(* Logix 5000 project; controller Generic 1768-L43 rev 15.6; software revision 15.01; part 3 of 10 *)
(* tags used below, declared in another part *)
   EL_CTRL_5 : UDT_AxisHistory_CTRL;
   EL_CTRL_6 : UDT_AxisHistory_CTRL;
   EventLog_N5 : UDT_AxisHistory_DLM[51];
   EventLog_N6 : UDT_AxisHistory_DLM[51];
   LogLength : DINT;
   Motion_Group : ALIAS FOR MotionGroup;
   Servo_Axis_Node_5 : ALIAS FOR AXIS_Servo_Generic;
   Servo_Axis_Node_6 : ALIAS FOR AXIS_Servo_Generic;
(* AXIS_EventLog, continued *)

ROUTINE R05_EventLog_Node5   (* ladder *)
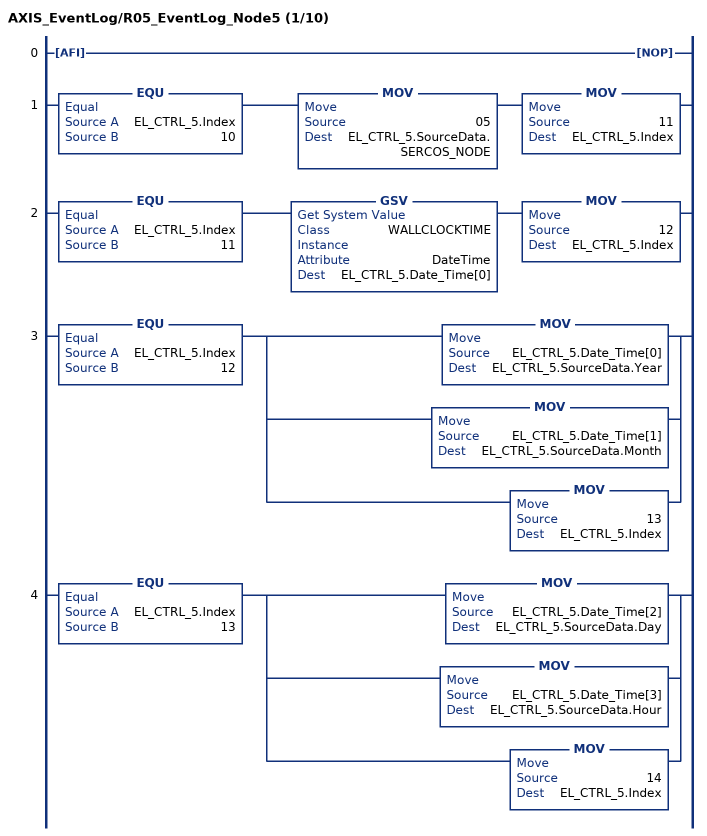
   0: AFI()NOP();
   1: EQU(EL_CTRL_5.Index,10)MOV(05,EL_CTRL_5.SourceData.SERCOS_NODE)MOV(11,EL_CTRL_5.Index);
   2: EQU(EL_CTRL_5.Index,11)GSV(WALLCLOCKTIME,,DateTime,EL_CTRL_5.Date_Time[0])MOV(12,EL_CTRL_5.Index);
   3: EQU(EL_CTRL_5.Index,12)[MOV(EL_CTRL_5.Date_Time[0],EL_CTRL_5.SourceData.Year) ,MOV(EL_CTRL_5.Date_Time[1],EL_CTRL_5.SourceData.Month) ,MOV(13,EL_CTRL_5.Index) ];
   4: EQU(EL_CTRL_5.Index,13)[MOV(EL_CTRL_5.Date_Time[2],EL_CTRL_5.SourceData.Day) ,MOV(EL_CTRL_5.Date_Time[3],EL_CTRL_5.SourceData.Hour) ,MOV(14,EL_CTRL_5.Index) ];
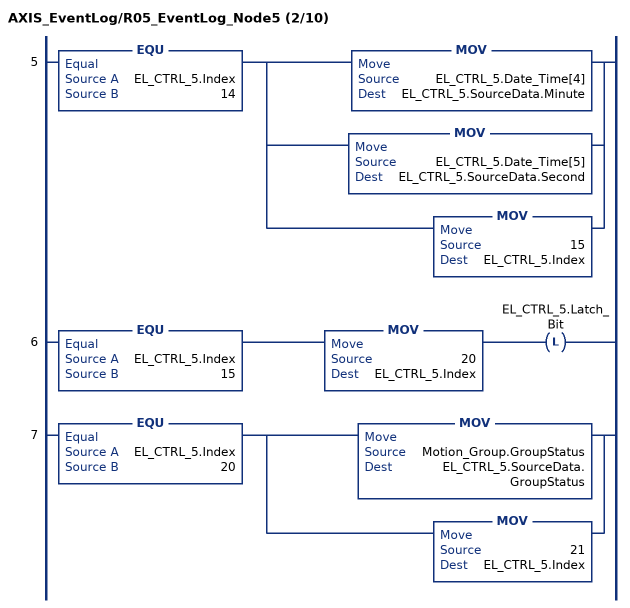
   5: EQU(EL_CTRL_5.Index,14)[MOV(EL_CTRL_5.Date_Time[4],EL_CTRL_5.SourceData.Minute) ,MOV(EL_CTRL_5.Date_Time[5],EL_CTRL_5.SourceData.Second) ,MOV(15,EL_CTRL_5.Index) ];
   6: EQU(EL_CTRL_5.Index,15)MOV(20,EL_CTRL_5.Index)OTL(EL_CTRL_5.Latch_Bit);
   7: EQU(EL_CTRL_5.Index,20)[MOV(Motion_Group.GroupStatus,EL_CTRL_5.SourceData.GroupStatus) ,MOV(21,EL_CTRL_5.Index) ];
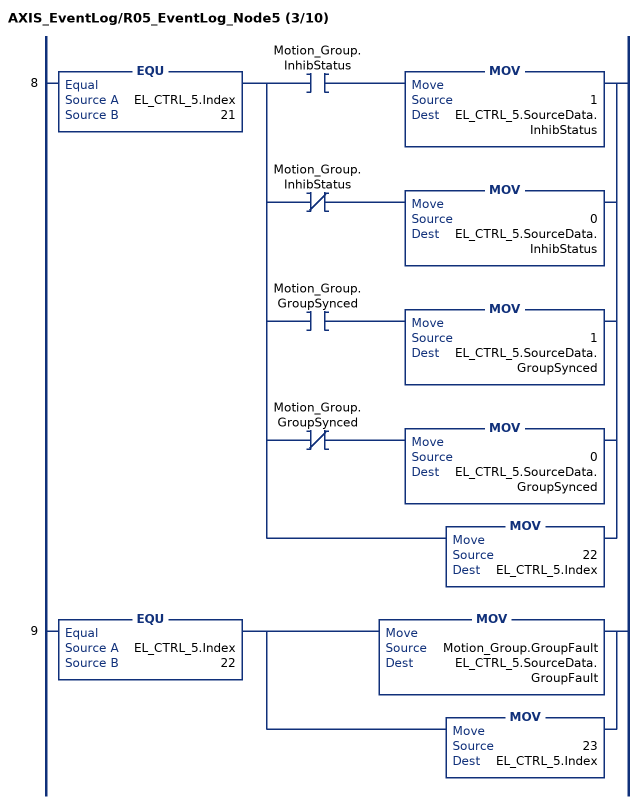
   8: EQU(EL_CTRL_5.Index,21)[XIC(Motion_Group.InhibStatus) MOV(1,EL_CTRL_5.SourceData.InhibStatus) ,XIO(Motion_Group.InhibStatus) MOV(0,EL_CTRL_5.SourceData.InhibStatus) ,XIC(Motion_Group.GroupSynced) MOV(1,EL_CTRL_5.SourceData.GroupSynced) ,XIO(Motion_Group.GroupSynced) MOV(0,EL_CTRL_5.SourceData.GroupSynced) ,MOV(22,EL_CTRL_5.Index) ];
   9: EQU(EL_CTRL_5.Index,22)[MOV(Motion_Group.GroupFault,EL_CTRL_5.SourceData.GroupFault) ,MOV(23,EL_CTRL_5.Index) ];
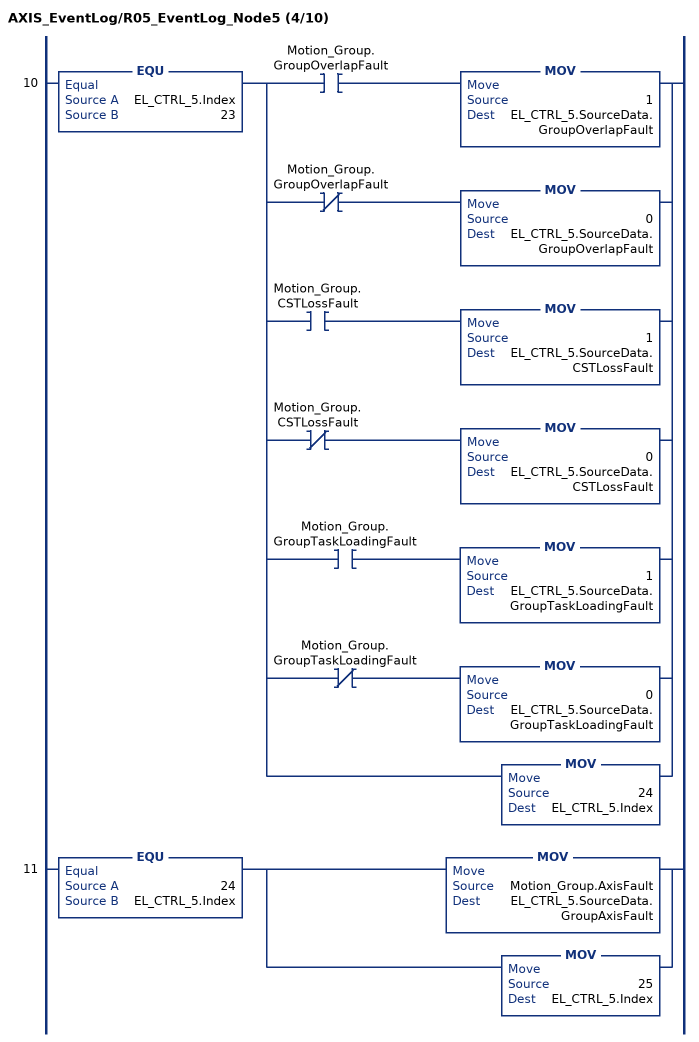
   10: EQU(EL_CTRL_5.Index,23)[XIC(Motion_Group.GroupOverlapFault) MOV(1,EL_CTRL_5.SourceData.GroupOverlapFault) ,XIO(Motion_Group.GroupOverlapFault) MOV(0,EL_CTRL_5.SourceData.GroupOverlapFault) ,XIC(Motion_Group.CSTLossFault) MOV(1,EL_CTRL_5.SourceData.CSTLossFault) ,XIO(Motion_Group.CSTLossFault) MOV(0,EL_CTRL_5.SourceData.CSTLossFault) ,XIC(Motion_Group.GroupTaskLoadingFault) MOV(1,EL_CTRL_5.SourceData.GroupTaskLoadingFault) ,XIO(Motion_Group.GroupTaskLoadingFault) MOV(0,EL_CTRL_5.SourceData.GroupTaskLoadingFault) ,MOV(24,EL_CTRL_5.Index) ];
   11: EQU(24,EL_CTRL_5.Index)[MOV(Motion_Group.AxisFault,EL_CTRL_5.SourceData.GroupAxisFault) ,MOV(25,EL_CTRL_5.Index) ];
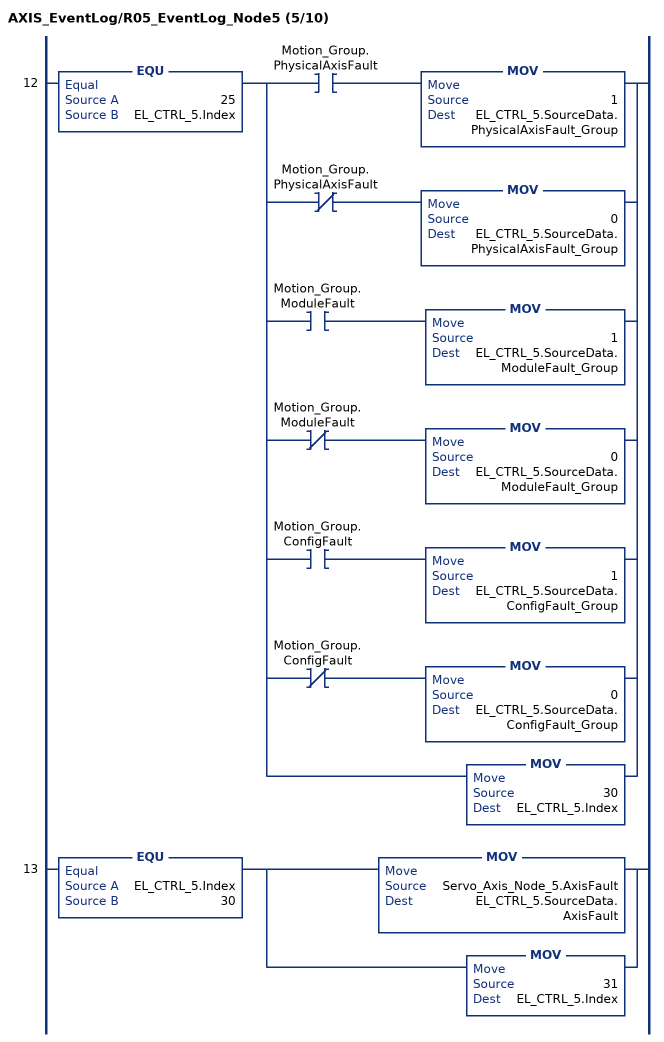
   12: EQU(25,EL_CTRL_5.Index)[XIC(Motion_Group.PhysicalAxisFault) MOV(1,EL_CTRL_5.SourceData.PhysicalAxisFault_Group) ,XIO(Motion_Group.PhysicalAxisFault) MOV(0,EL_CTRL_5.SourceData.PhysicalAxisFault_Group) ,XIC(Motion_Group.ModuleFault) MOV(1,EL_CTRL_5.SourceData.ModuleFault_Group) ,XIO(Motion_Group.ModuleFault) MOV(0,EL_CTRL_5.SourceData.ModuleFault_Group) ,XIC(Motion_Group.ConfigFault) MOV(1,EL_CTRL_5.SourceData.ConfigFault_Group) ,XIO(Motion_Group.ConfigFault) MOV(0,EL_CTRL_5.SourceData.ConfigFault_Group) ,MOV(30,EL_CTRL_5.Index) ];
   13: EQU(EL_CTRL_5.Index,30)[MOV(Servo_Axis_Node_5.AxisFault,EL_CTRL_5.SourceData.AxisFault) ,MOV(31,EL_CTRL_5.Index) ];
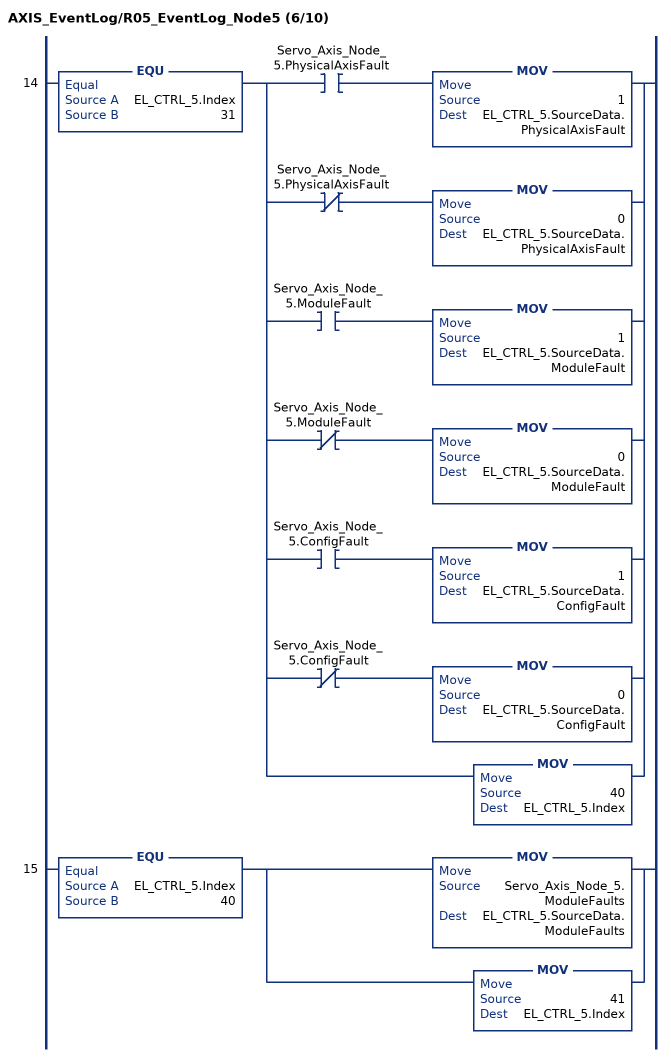
   14: EQU(EL_CTRL_5.Index,31)[XIC(Servo_Axis_Node_5.PhysicalAxisFault) MOV(1,EL_CTRL_5.SourceData.PhysicalAxisFault) ,XIO(Servo_Axis_Node_5.PhysicalAxisFault) MOV(0,EL_CTRL_5.SourceData.PhysicalAxisFault) ,XIC(Servo_Axis_Node_5.ModuleFault) MOV(1,EL_CTRL_5.SourceData.ModuleFault) ,XIO(Servo_Axis_Node_5.ModuleFault) MOV(0,EL_CTRL_5.SourceData.ModuleFault) ,XIC(Servo_Axis_Node_5.ConfigFault) MOV(1,EL_CTRL_5.SourceData.ConfigFault) ,XIO(Servo_Axis_Node_5.ConfigFault) MOV(0,EL_CTRL_5.SourceData.ConfigFault) ,MOV(40,EL_CTRL_5.Index) ];
   15: EQU(EL_CTRL_5.Index,40)[MOV(Servo_Axis_Node_5.ModuleFaults,EL_CTRL_5.SourceData.ModuleFaults) ,MOV(41,EL_CTRL_5.Index) ];
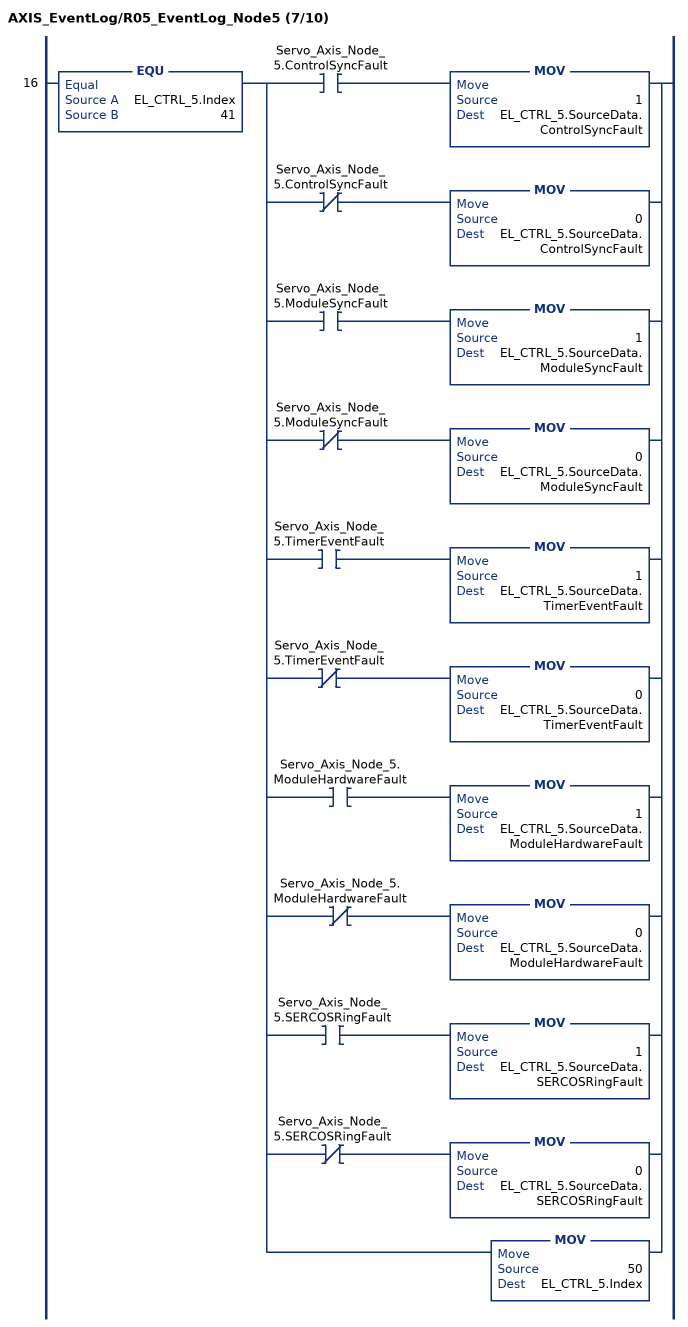
   16: EQU(EL_CTRL_5.Index,41)[XIC(Servo_Axis_Node_5.ControlSyncFault) MOV(1,EL_CTRL_5.SourceData.ControlSyncFault) ,XIO(Servo_Axis_Node_5.ControlSyncFault) MOV(0,EL_CTRL_5.SourceData.ControlSyncFault) ,XIC(Servo_Axis_Node_5.ModuleSyncFault) MOV(1,EL_CTRL_5.SourceData.ModuleSyncFault) ,XIO(Servo_Axis_Node_5.ModuleSyncFault) MOV(0,EL_CTRL_5.SourceData.ModuleSyncFault) ,XIC(Servo_Axis_Node_5.TimerEventFault) MOV(1,EL_CTRL_5.SourceData.TimerEventFault) ,XIO(Servo_Axis_Node_5.TimerEventFault) MOV(0,EL_CTRL_5.SourceData.TimerEventFault) ,XIC(Servo_Axis_Node_5.ModuleHardwareFault) MOV(1,EL_CTRL_5.SourceData.ModuleHardwareFault) ,XIO(Servo_Axis_Node_5.ModuleHardwareFault) MOV(0,EL_CTRL_5.SourceData.ModuleHardwareFault) ,XIC(Servo_Axis_Node_5.SERCOSRingFault) MOV(1,EL_CTRL_5.SourceData.SERCOSRingFault) ,XIO(Servo_Axis_Node_5.SERCOSRingFault) MOV(0,EL_CTRL_5.SourceData.SERCOSRingFault) ,MOV(50,EL_CTRL_5.Index) ];
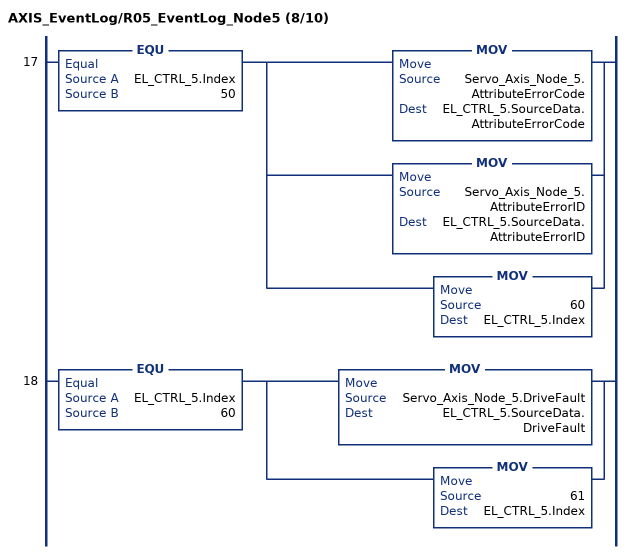
   17: EQU(EL_CTRL_5.Index,50)[MOV(Servo_Axis_Node_5.AttributeErrorCode,EL_CTRL_5.SourceData.AttributeErrorCode) ,MOV(Servo_Axis_Node_5.AttributeErrorID,EL_CTRL_5.SourceData.AttributeErrorID) ,MOV(60,EL_CTRL_5.Index) ];
   18: EQU(EL_CTRL_5.Index,60)[MOV(Servo_Axis_Node_5.DriveFault,EL_CTRL_5.SourceData.DriveFault) ,MOV(61,EL_CTRL_5.Index) ];
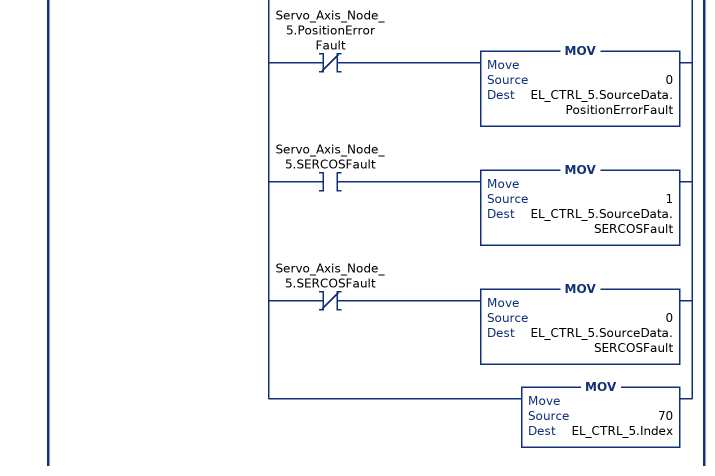
   19: EQU(EL_CTRL_5.Index,61)[XIC(Servo_Axis_Node_5.PosSoftOvertravelFault) MOV(1,EL_CTRL_5.SourceData.PosSoftOvertravelFault) ,XIO(Servo_Axis_Node_5.PosSoftOvertravelFault) MOV(0,EL_CTRL_5.SourceData.PosSoftOvertravelFault) ,XIC(Servo_Axis_Node_5.NegSoftOvertravelFault) MOV(1,EL_CTRL_5.SourceData.NegSoftOvertravelFault) ,XIO(Servo_Axis_Node_5.NegSoftOvertravelFault) MOV(0,EL_CTRL_5.SourceData.NegSoftOvertravelFault) ,XIC(Servo_Axis_Node_5.PosHardOvertravelFault) MOV(1,EL_CTRL_5.SourceData.PosHardOvertravelFault) ,XIO(Servo_Axis_Node_5.PosHardOvertravelFault) MOV(0,EL_CTRL_5.SourceData.PosHardOvertravelFault) ,XIC(Servo_Axis_Node_5.NegHardOvertravelFault) MOV(1,EL_CTRL_5.SourceData.NegHardOvertravelFault) ,XIO(Servo_Axis_Node_5.NegHardOvertravelFault) MOV(0,EL_CTRL_5.SourceData.NegHardOvertravelFault) ,XIC(Servo_Axis_Node_5.MotFeedbackFault) MOV(1,EL_CTRL_5.SourceData.MotFeedbackFault) ,XIO(Servo_Axis_Node_5.MotFeedbackFault) MOV(0,EL_CTRL_5.SourceData.MotFeedbackFault) ,XIC(Servo_Axis_Node_5.MotFeedbackNoiseFault) MOV(1,EL_CTRL_5.SourceData.MotFeedbackNoiseFault) ,XIO(Servo_Axis_Node_5.MotFeedbackNoiseFault) MOV(0,EL_CTRL_5.SourceData.MotFeedbackNoiseFault) ,XIC(Servo_Axis_Node_5.AuxFeedbackFault) MOV(1,EL_CTRL_5.SourceData.AuxFeedbackFault) ,XIO(Servo_Axis_Node_5.AuxFeedbackFault) MOV(0,EL_CTRL_5.SourceData.AuxFeedbackFault) ,XIC(Servo_Axis_Node_5.AuxFeedbackNoiseFault) MOV(1,EL_CTRL_5.SourceData.AuxFeedbackNoiseFault) ,XIO(Servo_Axis_Node_5.AuxFeedbackNoiseFault) MOV(0,EL_CTRL_5.SourceData.AuxFeedbackNoiseFault) ,XIC(Servo_Axis_Node_5.DriveEnableInputFault) MOV(1,EL_CTRL_5.SourceData.DriveEnableInputFault) ,XIO(Servo_Axis_Node_5.DriveEnableInputFault) MOV(0,EL_CTRL_5.SourceData.DriveEnableInputFault) ,XIC(Servo_Axis_Node_5.CommonBusFault) MOV(1,EL_CTRL_5.SourceData.CommonBusFault) ,XIO(Servo_Axis_Node_5.CommonBusFault) MOV(0,EL_CTRL_5.SourceData.CommonBusFault) ,XIC(Servo_Axis_Node_5.PreChargeOverloadFault) MOV(1,EL_CTRL_5.SourceData.PreChargeOverloadFault) ,XIO(Servo_Axis_Node_5.PreChargeOverloadFault) MOV(0,EL_CTRL_5.SourceData.PreChargeOverloadFault) ,XIC(Servo_Axis_Node_5.GroundShortFault) MOV(1,EL_CTRL_5.SourceData.GroundShortFault) ,XIO(Servo_Axis_Node_5.GroundShortFault) MOV(0,EL_CTRL_5.SourceData.GroundShortFault) ,XIC(Servo_Axis_Node_5.DriveHardFault) MOV(1,EL_CTRL_5.SourceData.DriveHardFault) ,XIO(Servo_Axis_Node_5.DriveHardFault) MOV(0,EL_CTRL_5.SourceData.DriveHardFault) ,XIC(Servo_Axis_Node_5.OverSpeedFault) MOV(1,EL_CTRL_5.SourceData.OverSpeedFault) ,XIO(Servo_Axis_Node_5.OverSpeedFault) MOV(0,EL_CTRL_5.SourceData.OverSpeedFault) ,XIC(Servo_Axis_Node_5.OverloadFault) MOV(1,EL_CTRL_5.SourceData.OverloadFault) ,XIO(Servo_Axis_Node_5.OverloadFault) MOV(0,EL_CTRL_5.SourceData.OverloadFault) ,XIC(Servo_Axis_Node_5.DriveOvertempFault) MOV(1,EL_CTRL_5.SourceData.DriveOvertempFault) ,XIO(Servo_Axis_Node_5.DriveOvertempFault) MOV(0,EL_CTRL_5.SourceData.DriveOvertempFault) ,XIC(Servo_Axis_Node_5.MotorOvertempFault) MOV(1,EL_CTRL_5.SourceData.MotorOvertempFault) ,XIO(Servo_Axis_Node_5.MotorOvertempFault) MOV(0,EL_CTRL_5.SourceData.MotorOvertempFault) ,XIC(Servo_Axis_Node_5.DriveCoolingFault) MOV(1,EL_CTRL_5.SourceData.DriveCoolingFault) ,XIO(Servo_Axis_Node_5.DriveCoolingFault) MOV(0,EL_CTRL_5.SourceData.DriveCoolingFault) ,XIC(Servo_Axis_Node_5.DriveControlVoltageFault) MOV(1,EL_CTRL_5.SourceData.DriveControlVoltageFault) ,XIO(Servo_Axis_Node_5.DriveControlVoltageFault) MOV(0,EL_CTRL_5.SourceData.DriveControlVoltageFault) ,XIC(Servo_Axis_Node_5.FeedbackFault) MOV(1,EL_CTRL_5.SourceData.FeedbackFault) ,XIO(Servo_Axis_Node_5.FeedbackFault) MOV(0,EL_CTRL_5.SourceData.FeedbackFault) ,XIC(Servo_Axis_Node_5.CommutationFault) MOV(1,EL_CTRL_5.SourceData.CommutationFault) ,XIO(Servo_Axis_Node_5.CommutationFault) MOV(0,EL_CTRL_5.SourceData.CommutationFault) ,XIC(Servo_Axis_Node_5.DriveOvercurrentFault) MOV(1,EL_CTRL_5.SourceData.DriveOvercurrentFault) ,XIO(Servo_Axis_Node_5.DriveOvercurrentFault) MOV(0,EL_CTRL_5.SourceData.DriveOvercurrentFault) ,XIC(Servo_Axis_Node_5.DriveOvervoltageFault) MOV(1,EL_CTRL_5.SourceData.DriveOvervoltageFault) ,XIO(Servo_Axis_Node_5.DriveOvervoltageFault) MOV(0,EL_CTRL_5.SourceData.DriveOvervoltageFault) ,XIC(Servo_Axis_Node_5.DriveUndervoltageFault) MOV(1,EL_CTRL_5.SourceData.DriveUndervoltageFault) ,XIO(Servo_Axis_Node_5.DriveUndervoltageFault) MOV(0,EL_CTRL_5.SourceData.DriveUndervoltageFault) ,XIC(Servo_Axis_Node_5.PowerPhaseLossFault) MOV(1,EL_CTRL_5.SourceData.PowerPhaseLossFault) ,XIO(Servo_Axis_Node_5.PowerPhaseLossFault) MOV(0,EL_CTRL_5.SourceData.PowerPhaseLossFault) ,XIC(Servo_Axis_Node_5.PositionErrorFault) MOV(1,EL_CTRL_5.SourceData.PositionErrorFault) ,XIO(Servo_Axis_Node_5.PositionErrorFault) MOV(0,EL_CTRL_5.SourceData.PositionErrorFault) ,XIC(Servo_Axis_Node_5.SERCOSFault) MOV(1,EL_CTRL_5.SourceData.SERCOSFault) ,XIO(Servo_Axis_Node_5.SERCOSFault) MOV(0,EL_CTRL_5.SourceData.SERCOSFault) ,MOV(70,EL_CTRL_5.Index) ];
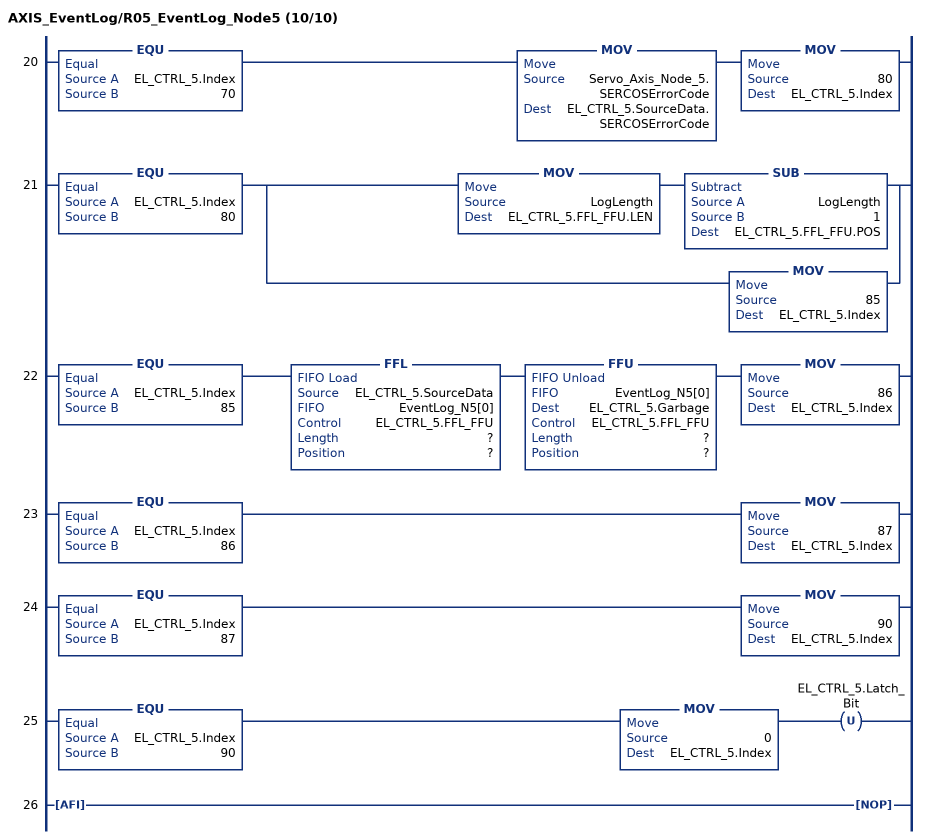
   20: EQU(EL_CTRL_5.Index,70)MOV(Servo_Axis_Node_5.SERCOSErrorCode,EL_CTRL_5.SourceData.SERCOSErrorCode)MOV(80,EL_CTRL_5.Index);
   21: EQU(EL_CTRL_5.Index,80)[MOV(LogLength,EL_CTRL_5.FFL_FFU.LEN) SUB(LogLength,1,EL_CTRL_5.FFL_FFU.POS) ,MOV(85,EL_CTRL_5.Index) ];
   22: EQU(EL_CTRL_5.Index,85)FFL(EL_CTRL_5.SourceData,EventLog_N5[0],EL_CTRL_5.FFL_FFU,?,?)FFU(EventLog_N5[0],EL_CTRL_5.Garbage,EL_CTRL_5.FFL_FFU,?,?)MOV(86,EL_CTRL_5.Index);
   23: EQU(EL_CTRL_5.Index,86)MOV(87,EL_CTRL_5.Index);
   24: EQU(EL_CTRL_5.Index,87)MOV(90,EL_CTRL_5.Index);
   25: EQU(EL_CTRL_5.Index,90)MOV(0,EL_CTRL_5.Index)OTU(EL_CTRL_5.Latch_Bit);
   26: AFI()NOP();
END_ROUTINE

ROUTINE R06_EventLog_Node6   (* ladder *)
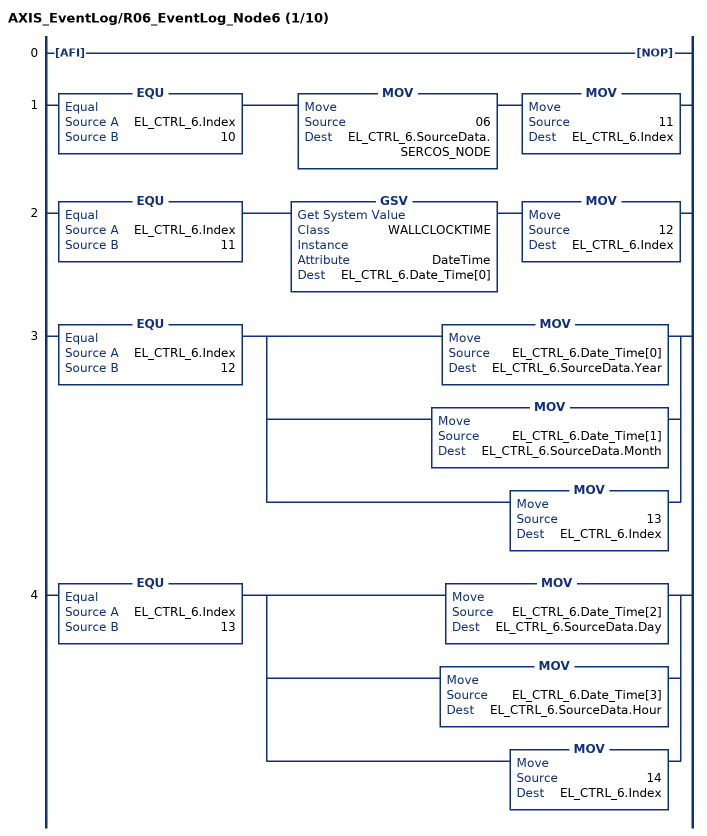
   0: AFI()NOP();
   1: EQU(EL_CTRL_6.Index,10)MOV(06,EL_CTRL_6.SourceData.SERCOS_NODE)MOV(11,EL_CTRL_6.Index);
   2: EQU(EL_CTRL_6.Index,11)GSV(WALLCLOCKTIME,,DateTime,EL_CTRL_6.Date_Time[0])MOV(12,EL_CTRL_6.Index);
   3: EQU(EL_CTRL_6.Index,12)[MOV(EL_CTRL_6.Date_Time[0],EL_CTRL_6.SourceData.Year) ,MOV(EL_CTRL_6.Date_Time[1],EL_CTRL_6.SourceData.Month) ,MOV(13,EL_CTRL_6.Index) ];
   4: EQU(EL_CTRL_6.Index,13)[MOV(EL_CTRL_6.Date_Time[2],EL_CTRL_6.SourceData.Day) ,MOV(EL_CTRL_6.Date_Time[3],EL_CTRL_6.SourceData.Hour) ,MOV(14,EL_CTRL_6.Index) ];
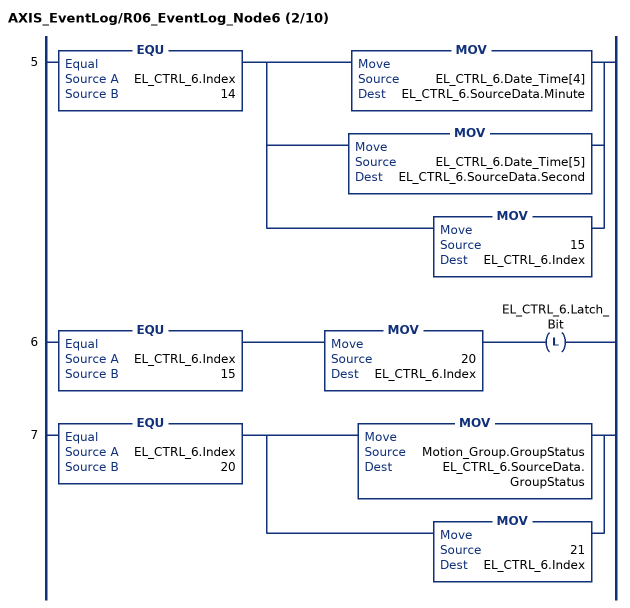
   5: EQU(EL_CTRL_6.Index,14)[MOV(EL_CTRL_6.Date_Time[4],EL_CTRL_6.SourceData.Minute) ,MOV(EL_CTRL_6.Date_Time[5],EL_CTRL_6.SourceData.Second) ,MOV(15,EL_CTRL_6.Index) ];
   6: EQU(EL_CTRL_6.Index,15)MOV(20,EL_CTRL_6.Index)OTL(EL_CTRL_6.Latch_Bit);
   7: EQU(EL_CTRL_6.Index,20)[MOV(Motion_Group.GroupStatus,EL_CTRL_6.SourceData.GroupStatus) ,MOV(21,EL_CTRL_6.Index) ];
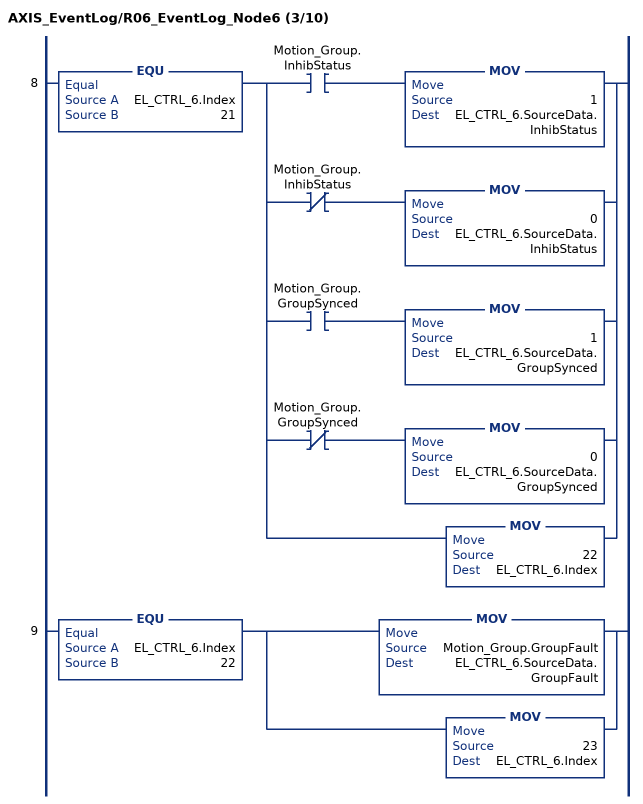
   8: EQU(EL_CTRL_6.Index,21)[XIC(Motion_Group.InhibStatus) MOV(1,EL_CTRL_6.SourceData.InhibStatus) ,XIO(Motion_Group.InhibStatus) MOV(0,EL_CTRL_6.SourceData.InhibStatus) ,XIC(Motion_Group.GroupSynced) MOV(1,EL_CTRL_6.SourceData.GroupSynced) ,XIO(Motion_Group.GroupSynced) MOV(0,EL_CTRL_6.SourceData.GroupSynced) ,MOV(22,EL_CTRL_6.Index) ];
   9: EQU(EL_CTRL_6.Index,22)[MOV(Motion_Group.GroupFault,EL_CTRL_6.SourceData.GroupFault) ,MOV(23,EL_CTRL_6.Index) ];
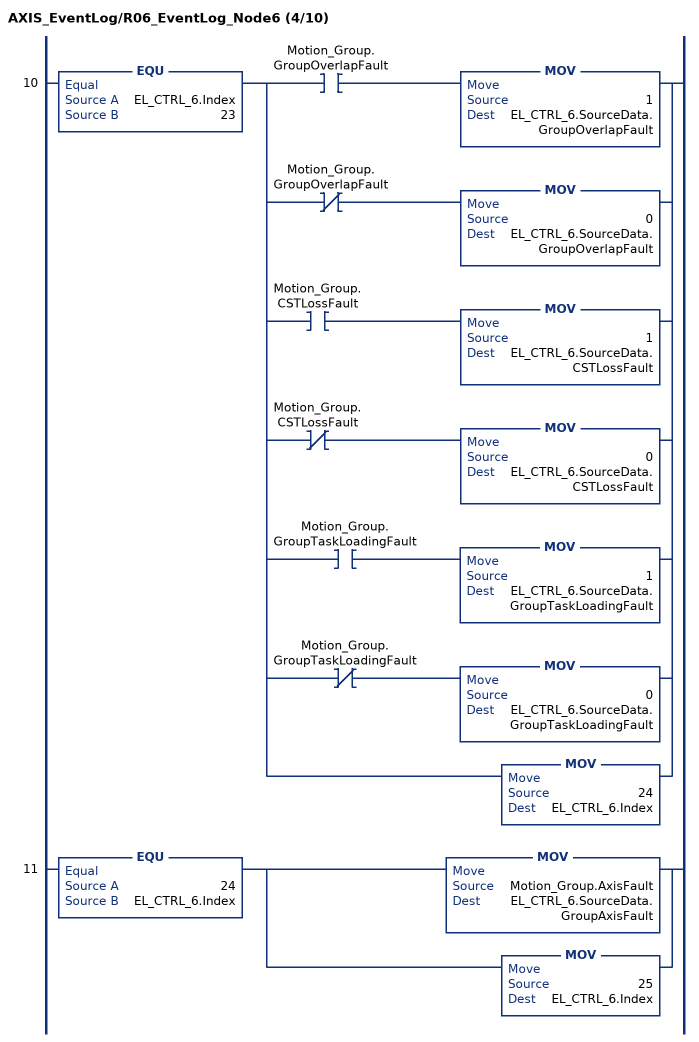
   10: EQU(EL_CTRL_6.Index,23)[XIC(Motion_Group.GroupOverlapFault) MOV(1,EL_CTRL_6.SourceData.GroupOverlapFault) ,XIO(Motion_Group.GroupOverlapFault) MOV(0,EL_CTRL_6.SourceData.GroupOverlapFault) ,XIC(Motion_Group.CSTLossFault) MOV(1,EL_CTRL_6.SourceData.CSTLossFault) ,XIO(Motion_Group.CSTLossFault) MOV(0,EL_CTRL_6.SourceData.CSTLossFault) ,XIC(Motion_Group.GroupTaskLoadingFault) MOV(1,EL_CTRL_6.SourceData.GroupTaskLoadingFault) ,XIO(Motion_Group.GroupTaskLoadingFault) MOV(0,EL_CTRL_6.SourceData.GroupTaskLoadingFault) ,MOV(24,EL_CTRL_6.Index) ];
   11: EQU(24,EL_CTRL_6.Index)[MOV(Motion_Group.AxisFault,EL_CTRL_6.SourceData.GroupAxisFault) ,MOV(25,EL_CTRL_6.Index) ];
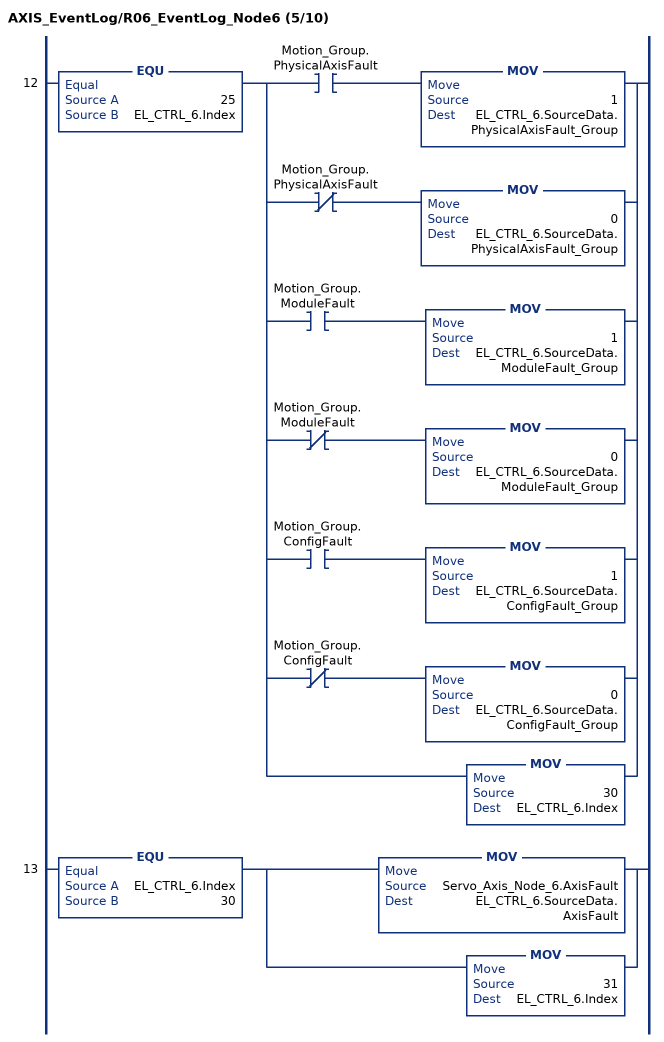
   12: EQU(25,EL_CTRL_6.Index)[XIC(Motion_Group.PhysicalAxisFault) MOV(1,EL_CTRL_6.SourceData.PhysicalAxisFault_Group) ,XIO(Motion_Group.PhysicalAxisFault) MOV(0,EL_CTRL_6.SourceData.PhysicalAxisFault_Group) ,XIC(Motion_Group.ModuleFault) MOV(1,EL_CTRL_6.SourceData.ModuleFault_Group) ,XIO(Motion_Group.ModuleFault) MOV(0,EL_CTRL_6.SourceData.ModuleFault_Group) ,XIC(Motion_Group.ConfigFault) MOV(1,EL_CTRL_6.SourceData.ConfigFault_Group) ,XIO(Motion_Group.ConfigFault) MOV(0,EL_CTRL_6.SourceData.ConfigFault_Group) ,MOV(30,EL_CTRL_6.Index) ];
   13: EQU(EL_CTRL_6.Index,30)[MOV(Servo_Axis_Node_6.AxisFault,EL_CTRL_6.SourceData.AxisFault) ,MOV(31,EL_CTRL_6.Index) ];
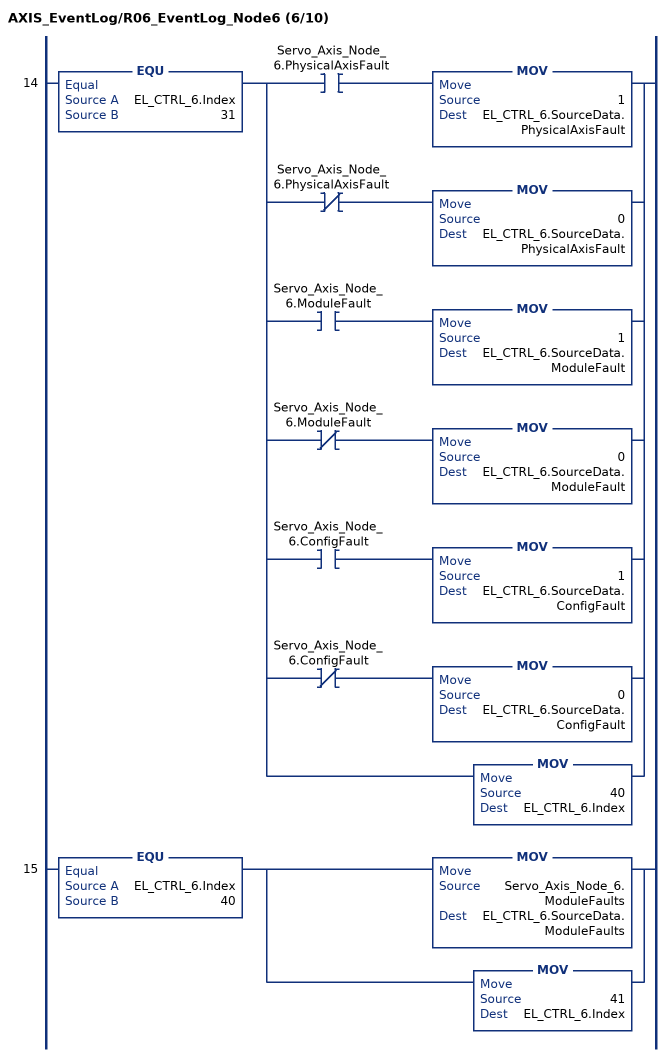
   14: EQU(EL_CTRL_6.Index,31)[XIC(Servo_Axis_Node_6.PhysicalAxisFault) MOV(1,EL_CTRL_6.SourceData.PhysicalAxisFault) ,XIO(Servo_Axis_Node_6.PhysicalAxisFault) MOV(0,EL_CTRL_6.SourceData.PhysicalAxisFault) ,XIC(Servo_Axis_Node_6.ModuleFault) MOV(1,EL_CTRL_6.SourceData.ModuleFault) ,XIO(Servo_Axis_Node_6.ModuleFault) MOV(0,EL_CTRL_6.SourceData.ModuleFault) ,XIC(Servo_Axis_Node_6.ConfigFault) MOV(1,EL_CTRL_6.SourceData.ConfigFault) ,XIO(Servo_Axis_Node_6.ConfigFault) MOV(0,EL_CTRL_6.SourceData.ConfigFault) ,MOV(40,EL_CTRL_6.Index) ];
   15: EQU(EL_CTRL_6.Index,40)[MOV(Servo_Axis_Node_6.ModuleFaults,EL_CTRL_6.SourceData.ModuleFaults) ,MOV(41,EL_CTRL_6.Index) ];
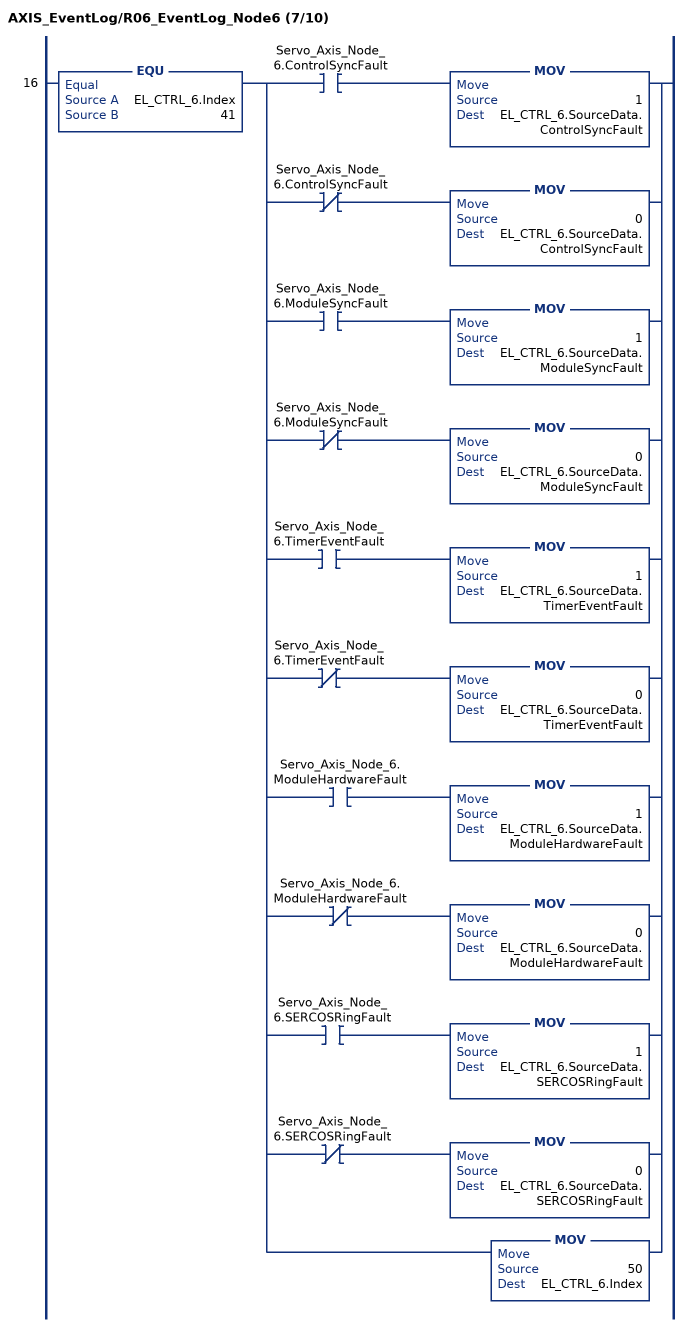
   16: EQU(EL_CTRL_6.Index,41)[XIC(Servo_Axis_Node_6.ControlSyncFault) MOV(1,EL_CTRL_6.SourceData.ControlSyncFault) ,XIO(Servo_Axis_Node_6.ControlSyncFault) MOV(0,EL_CTRL_6.SourceData.ControlSyncFault) ,XIC(Servo_Axis_Node_6.ModuleSyncFault) MOV(1,EL_CTRL_6.SourceData.ModuleSyncFault) ,XIO(Servo_Axis_Node_6.ModuleSyncFault) MOV(0,EL_CTRL_6.SourceData.ModuleSyncFault) ,XIC(Servo_Axis_Node_6.TimerEventFault) MOV(1,EL_CTRL_6.SourceData.TimerEventFault) ,XIO(Servo_Axis_Node_6.TimerEventFault) MOV(0,EL_CTRL_6.SourceData.TimerEventFault) ,XIC(Servo_Axis_Node_6.ModuleHardwareFault) MOV(1,EL_CTRL_6.SourceData.ModuleHardwareFault) ,XIO(Servo_Axis_Node_6.ModuleHardwareFault) MOV(0,EL_CTRL_6.SourceData.ModuleHardwareFault) ,XIC(Servo_Axis_Node_6.SERCOSRingFault) MOV(1,EL_CTRL_6.SourceData.SERCOSRingFault) ,XIO(Servo_Axis_Node_6.SERCOSRingFault) MOV(0,EL_CTRL_6.SourceData.SERCOSRingFault) ,MOV(50,EL_CTRL_6.Index) ];
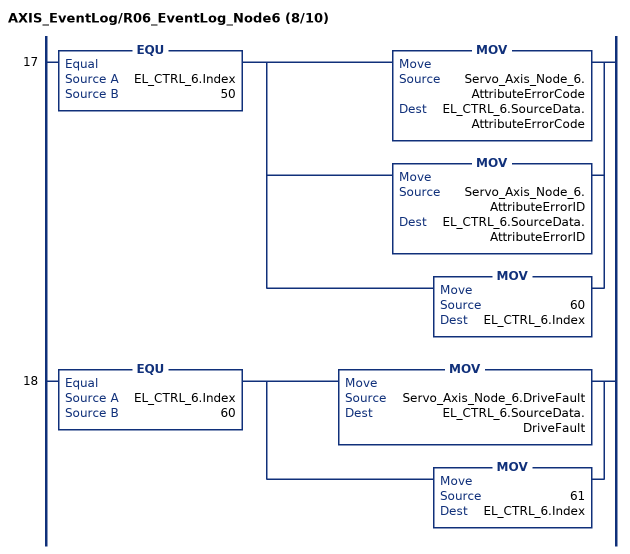
   17: EQU(EL_CTRL_6.Index,50)[MOV(Servo_Axis_Node_6.AttributeErrorCode,EL_CTRL_6.SourceData.AttributeErrorCode) ,MOV(Servo_Axis_Node_6.AttributeErrorID,EL_CTRL_6.SourceData.AttributeErrorID) ,MOV(60,EL_CTRL_6.Index) ];
   18: EQU(EL_CTRL_6.Index,60)[MOV(Servo_Axis_Node_6.DriveFault,EL_CTRL_6.SourceData.DriveFault) ,MOV(61,EL_CTRL_6.Index) ];
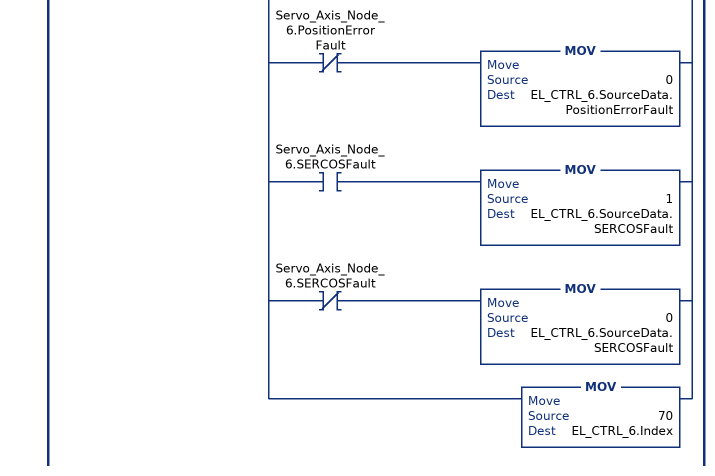
   19: EQU(EL_CTRL_6.Index,61)[XIC(Servo_Axis_Node_6.PosSoftOvertravelFault) MOV(1,EL_CTRL_6.SourceData.PosSoftOvertravelFault) ,XIO(Servo_Axis_Node_6.PosSoftOvertravelFault) MOV(0,EL_CTRL_6.SourceData.PosSoftOvertravelFault) ,XIC(Servo_Axis_Node_6.NegSoftOvertravelFault) MOV(1,EL_CTRL_6.SourceData.NegSoftOvertravelFault) ,XIO(Servo_Axis_Node_6.NegSoftOvertravelFault) MOV(0,EL_CTRL_6.SourceData.NegSoftOvertravelFault) ,XIC(Servo_Axis_Node_6.PosHardOvertravelFault) MOV(1,EL_CTRL_6.SourceData.PosHardOvertravelFault) ,XIO(Servo_Axis_Node_6.PosHardOvertravelFault) MOV(0,EL_CTRL_6.SourceData.PosHardOvertravelFault) ,XIC(Servo_Axis_Node_6.NegHardOvertravelFault) MOV(1,EL_CTRL_6.SourceData.NegHardOvertravelFault) ,XIO(Servo_Axis_Node_6.NegHardOvertravelFault) MOV(0,EL_CTRL_6.SourceData.NegHardOvertravelFault) ,XIC(Servo_Axis_Node_6.MotFeedbackFault) MOV(1,EL_CTRL_6.SourceData.MotFeedbackFault) ,XIO(Servo_Axis_Node_6.MotFeedbackFault) MOV(0,EL_CTRL_6.SourceData.MotFeedbackFault) ,XIC(Servo_Axis_Node_6.MotFeedbackNoiseFault) MOV(1,EL_CTRL_6.SourceData.MotFeedbackNoiseFault) ,XIO(Servo_Axis_Node_6.MotFeedbackNoiseFault) MOV(0,EL_CTRL_6.SourceData.MotFeedbackNoiseFault) ,XIC(Servo_Axis_Node_6.AuxFeedbackFault) MOV(1,EL_CTRL_6.SourceData.AuxFeedbackFault) ,XIO(Servo_Axis_Node_6.AuxFeedbackFault) MOV(0,EL_CTRL_6.SourceData.AuxFeedbackFault) ,XIC(Servo_Axis_Node_6.AuxFeedbackNoiseFault) MOV(1,EL_CTRL_6.SourceData.AuxFeedbackNoiseFault) ,XIO(Servo_Axis_Node_6.AuxFeedbackNoiseFault) MOV(0,EL_CTRL_6.SourceData.AuxFeedbackNoiseFault) ,XIC(Servo_Axis_Node_6.DriveEnableInputFault) MOV(1,EL_CTRL_6.SourceData.DriveEnableInputFault) ,XIO(Servo_Axis_Node_6.DriveEnableInputFault) MOV(0,EL_CTRL_6.SourceData.DriveEnableInputFault) ,XIC(Servo_Axis_Node_6.CommonBusFault) MOV(1,EL_CTRL_6.SourceData.CommonBusFault) ,XIO(Servo_Axis_Node_6.CommonBusFault) MOV(0,EL_CTRL_6.SourceData.CommonBusFault) ,XIC(Servo_Axis_Node_6.PreChargeOverloadFault) MOV(1,EL_CTRL_6.SourceData.PreChargeOverloadFault) ,XIO(Servo_Axis_Node_6.PreChargeOverloadFault) MOV(0,EL_CTRL_6.SourceData.PreChargeOverloadFault) ,XIC(Servo_Axis_Node_6.GroundShortFault) MOV(1,EL_CTRL_6.SourceData.GroundShortFault) ,XIO(Servo_Axis_Node_6.GroundShortFault) MOV(0,EL_CTRL_6.SourceData.GroundShortFault) ,XIC(Servo_Axis_Node_6.DriveHardFault) MOV(1,EL_CTRL_6.SourceData.DriveHardFault) ,XIO(Servo_Axis_Node_6.DriveHardFault) MOV(0,EL_CTRL_6.SourceData.DriveHardFault) ,XIC(Servo_Axis_Node_6.OverSpeedFault) MOV(1,EL_CTRL_6.SourceData.OverSpeedFault) ,XIO(Servo_Axis_Node_6.OverSpeedFault) MOV(0,EL_CTRL_6.SourceData.OverSpeedFault) ,XIC(Servo_Axis_Node_6.OverloadFault) MOV(1,EL_CTRL_6.SourceData.OverloadFault) ,XIO(Servo_Axis_Node_6.OverloadFault) MOV(0,EL_CTRL_6.SourceData.OverloadFault) ,XIC(Servo_Axis_Node_6.DriveOvertempFault) MOV(1,EL_CTRL_6.SourceData.DriveOvertempFault) ,XIO(Servo_Axis_Node_6.DriveOvertempFault) MOV(0,EL_CTRL_6.SourceData.DriveOvertempFault) ,XIC(Servo_Axis_Node_6.MotorOvertempFault) MOV(1,EL_CTRL_6.SourceData.MotorOvertempFault) ,XIO(Servo_Axis_Node_6.MotorOvertempFault) MOV(0,EL_CTRL_6.SourceData.MotorOvertempFault) ,XIC(Servo_Axis_Node_6.DriveCoolingFault) MOV(1,EL_CTRL_6.SourceData.DriveCoolingFault) ,XIO(Servo_Axis_Node_6.DriveCoolingFault) MOV(0,EL_CTRL_6.SourceData.DriveCoolingFault) ,XIC(Servo_Axis_Node_6.DriveControlVoltageFault) MOV(1,EL_CTRL_6.SourceData.DriveControlVoltageFault) ,XIO(Servo_Axis_Node_6.DriveControlVoltageFault) MOV(0,EL_CTRL_6.SourceData.DriveControlVoltageFault) ,XIC(Servo_Axis_Node_6.FeedbackFault) MOV(1,EL_CTRL_6.SourceData.FeedbackFault) ,XIO(Servo_Axis_Node_6.FeedbackFault) MOV(0,EL_CTRL_6.SourceData.FeedbackFault) ,XIC(Servo_Axis_Node_6.CommutationFault) MOV(1,EL_CTRL_6.SourceData.CommutationFault) ,XIO(Servo_Axis_Node_6.CommutationFault) MOV(0,EL_CTRL_6.SourceData.CommutationFault) ,XIC(Servo_Axis_Node_6.DriveOvercurrentFault) MOV(1,EL_CTRL_6.SourceData.DriveOvercurrentFault) ,XIO(Servo_Axis_Node_6.DriveOvercurrentFault) MOV(0,EL_CTRL_6.SourceData.DriveOvercurrentFault) ,XIC(Servo_Axis_Node_6.DriveOvervoltageFault) MOV(1,EL_CTRL_6.SourceData.DriveOvervoltageFault) ,XIO(Servo_Axis_Node_6.DriveOvervoltageFault) MOV(0,EL_CTRL_6.SourceData.DriveOvervoltageFault) ,XIC(Servo_Axis_Node_6.DriveUndervoltageFault) MOV(1,EL_CTRL_6.SourceData.DriveUndervoltageFault) ,XIO(Servo_Axis_Node_6.DriveUndervoltageFault) MOV(0,EL_CTRL_6.SourceData.DriveUndervoltageFault) ,XIC(Servo_Axis_Node_6.PowerPhaseLossFault) MOV(1,EL_CTRL_6.SourceData.PowerPhaseLossFault) ,XIO(Servo_Axis_Node_6.PowerPhaseLossFault) MOV(0,EL_CTRL_6.SourceData.PowerPhaseLossFault) ,XIC(Servo_Axis_Node_6.PositionErrorFault) MOV(1,EL_CTRL_6.SourceData.PositionErrorFault) ,XIO(Servo_Axis_Node_6.PositionErrorFault) MOV(0,EL_CTRL_6.SourceData.PositionErrorFault) ,XIC(Servo_Axis_Node_6.SERCOSFault) MOV(1,EL_CTRL_6.SourceData.SERCOSFault) ,XIO(Servo_Axis_Node_6.SERCOSFault) MOV(0,EL_CTRL_6.SourceData.SERCOSFault) ,MOV(70,EL_CTRL_6.Index) ];
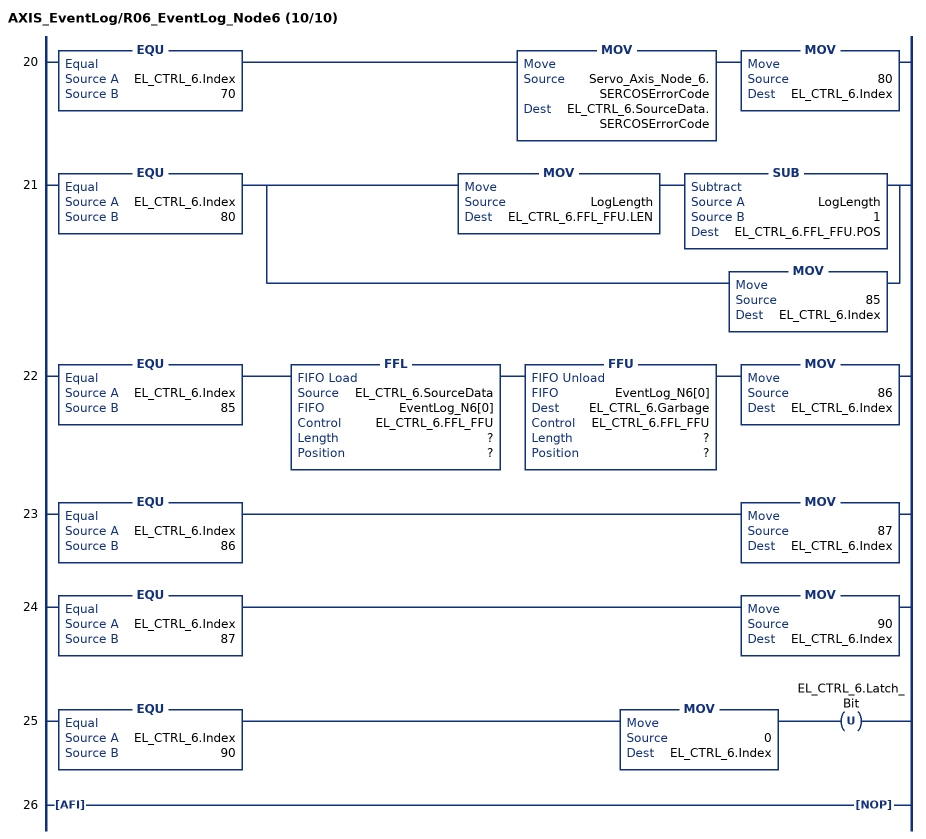
   20: EQU(EL_CTRL_6.Index,70)MOV(Servo_Axis_Node_6.SERCOSErrorCode,EL_CTRL_6.SourceData.SERCOSErrorCode)MOV(80,EL_CTRL_6.Index);
   21: EQU(EL_CTRL_6.Index,80)[MOV(LogLength,EL_CTRL_6.FFL_FFU.LEN) SUB(LogLength,1,EL_CTRL_6.FFL_FFU.POS) ,MOV(85,EL_CTRL_6.Index) ];
   22: EQU(EL_CTRL_6.Index,85)FFL(EL_CTRL_6.SourceData,EventLog_N6[0],EL_CTRL_6.FFL_FFU,?,?)FFU(EventLog_N6[0],EL_CTRL_6.Garbage,EL_CTRL_6.FFL_FFU,?,?)MOV(86,EL_CTRL_6.Index);
   23: EQU(EL_CTRL_6.Index,86)MOV(87,EL_CTRL_6.Index);
   24: EQU(EL_CTRL_6.Index,87)MOV(90,EL_CTRL_6.Index);
   25: EQU(EL_CTRL_6.Index,90)MOV(0,EL_CTRL_6.Index)OTU(EL_CTRL_6.Latch_Bit);
   26: AFI()NOP();
END_ROUTINE
